// TIA Portal V20 export
TYPE "Interlock_Cajas_PLC_IKPAL"
   STRUCT
      BitDeVida : Bool;
      Libre_01 : Bool;
      Libre_02 : Bool;
      Libre_03 : Bool;
      Libre_04 : Bool;
      Libre_05 : Bool;
      Libre_06 : Bool;
      Libre_07 : Bool;
      Cajas_Automatico : Bool;
      Cajas_Marcha : Bool;
      Cajas_Error : Bool;
      Libre_13 : Bool;
      Libre_14 : Bool;
      Libre_15 : Bool;
      Libre_16 : Bool;
      Libre_17 : Bool;
      Libre_20 : Bool;
      Libre_21 : Bool;
      Libre_22 : Bool;
      Libre_23 : Bool;
      Libre_24 : Bool;
      Libre_25 : Bool;
      Libre_26 : Bool;
      Libre_27 : Bool;
      Libre_30 : Bool;
      Libre_31 : Bool;
      Libre_32 : Bool;
      Libre_33 : Bool;
      Libre_34 : Bool;
      Libre_35 : Bool;
      Libre_36 : Bool;
      Libre_37 : Bool;
      AvisoCajas_PRV : Bool;
      Libre_41 : Bool;
      Libre_42 : Bool;
      Libre_43 : Bool;
      Libre_44 : Bool;
      Libre_45 : Bool;
      Libre_46 : Bool;
      Libre_47 : Bool;
      Libre_50 : Bool;
      Libre_51 : Bool;
      Libre_52 : Bool;
      Libre_53 : Bool;
      Libre_54 : Bool;
      Libre_55 : Bool;
      Libre_56 : Bool;
      Libre_57 : Bool;
   END_STRUCT;
END_TYPE
